// TIA Portal project "babu_fountain" (V15)

(* hardware
DEVICE "S7-1200 station_1"  S7-1200 Station
   slot 0: "Rack_0"  S7-1200 Rack  Rack  V1.0
   slot 1: "PLC_1"  CPU 1212C DC/DC/DC  6ES7 212-1AE40-0XB0  V4.2
*)

// ===== PLC "PLC_1"  CPU 1212C DC/DC/DC =====

VAR_GLOBAL   // PLC tag table "Tag table_1"
   "PUSH BUTTON" AT %M0.0 : Bool;
   "PUSH BUTTON MEMORY" AT %M0.1 : Bool;
   "HIGH SPRAY" AT %Q0.2 : Bool;
   "LOW SPRAY" AT %Q0.3 : Bool;
   "START" AT %M0.4 : Bool;
END_VAR

// folder: System blocks/Program resources

DATA_BLOCK "IEC_Timer_0_DB"   // DB1
{ S7_Optimized_Access := 'TRUE' }
AUTHOR : Simatic
FAMILY : IEC
NAME : IEC_TMR
VERSION : 1.0
// stored: InstanceOfName IEC_TIMER
"IEC_TIMER"
BEGIN
END_DATA_BLOCK

DATA_BLOCK "IEC_Timer_0_DB_1"   // DB2
{ S7_Optimized_Access := 'TRUE' }
AUTHOR : Simatic
FAMILY : IEC
NAME : IEC_TMR
VERSION : 1.0
// stored: InstanceOfName IEC_TIMER
"IEC_TIMER"
BEGIN
END_DATA_BLOCK

DATA_BLOCK "IEC_Timer_0_DB_2"   // DB3
{ S7_Optimized_Access := 'TRUE' }
AUTHOR : Simatic
FAMILY : IEC
NAME : IEC_TMR
VERSION : 1.0
// stored: InstanceOfName IEC_TIMER
"IEC_TIMER"
BEGIN
END_DATA_BLOCK

// folder: (top level)

ORGANIZATION_BLOCK "Main"   // OB1, LAD, ProgramCycle
TITLE = "Main Program Sweep (Cycle)"
{ S7_Optimized_Access := 'TRUE' }
VERSION : 0.1
   VAR_INPUT
      Initial_Call : Bool;   // Initial call of this OB
      Remanence : Bool;   // =True, if remanent data are available
   END_VAR
BEGIN

REGION Network 1
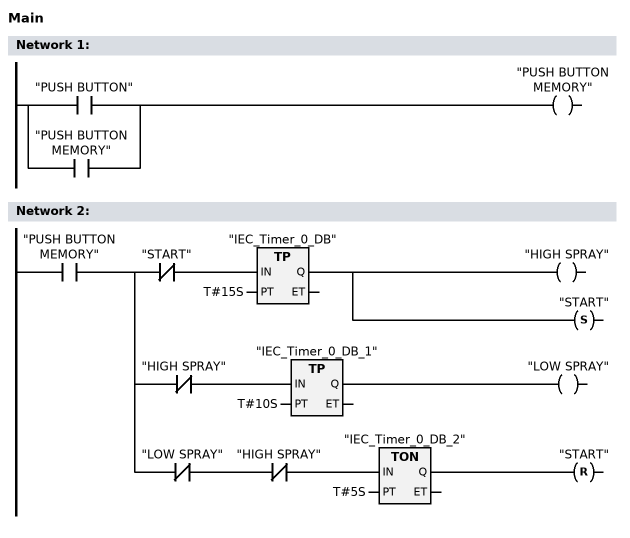
   RUNG wire#powerrail
      Contact( "PUSH BUTTON" )
      wire#w1
      Coil( "PUSH BUTTON MEMORY" )
   END_RUNG
   RUNG wire#powerrail
      Contact( "PUSH BUTTON MEMORY" )
   END_RUNG wire#w1
   // the same network as SCL:
   "PUSH BUTTON MEMORY" := "PUSH BUTTON" OR "PUSH BUTTON MEMORY";
END_REGION

REGION Network 2
   "IEC_Timer_0_DB".TP(IN := "PUSH BUTTON MEMORY" AND NOT "START", PT := T#15S);
   "HIGH SPRAY" := "IEC_Timer_0_DB".Q;
   IF "IEC_Timer_0_DB".Q THEN "START" := TRUE; END_IF;
   "IEC_Timer_0_DB_1".TP(IN := "PUSH BUTTON MEMORY" AND NOT "HIGH SPRAY", PT := T#10S);
   "LOW SPRAY" := "IEC_Timer_0_DB_1".Q;
   "IEC_Timer_0_DB_2".TON(IN := "PUSH BUTTON MEMORY" AND NOT "LOW SPRAY" AND NOT "HIGH SPRAY", PT := T#5S);
   IF "IEC_Timer_0_DB_2".Q THEN "START" := FALSE; END_IF;
END_REGION
END_ORGANIZATION_BLOCK